FUNCTION_BLOCK FB_V1_C1_Virtual_Input_Source IMPLEMENTS I_VirtualInputSource, I_V1_Virtual_Input_Source
VAR
	_fbSource: I_InputSource;
	
	_nSourceClientID: LWORD;
	_nDataHandle: ULINT;
	_nElements: UDINT;
	
	_nSelectedElement: UDINT;
	_nSelectedOversample: UDINT;
	
	_nContext: DWORD;
	_stInputs: ST_T1_Inputs;
	
	_nTimestamp: ULINT;
END_VAR

PROPERTY bEndOfData : BOOL
GET
bEndOfData:= _nElements = 0 OR (_nSelectedElement >= _nElements AND _nSelectedOversample >= _fbSource.nMaxOversamplingFactor);
END_GET
END_PROPERTY

METHOD Done : BOOL
VAR
END_VAR
IF bEndOfData AND _nElements > 0 THEN
	_nElements:= 0;
	_fbSource.ClientDone(_nSourceClientID);
END_IF

_nContext:= 0;
END_METHOD

PROPERTY dtTimestamp : DCTIMESTRUCT
GET
dtTimestamp:= F_AlyTimestampToDCTimestruct(_nTimestamp);
END_GET
END_PROPERTY

PROPERTY eSourceState : E_DataSourceState
GET
eSourceState:= _fbSource.eDataState;
END_GET
END_PROPERTY

METHOD FB_init : BOOL
VAR_INPUT
	bInitRetains: BOOL; // if TRUE, the retain variables are initialized (warm start / cold start)
	bInCopyCode: BOOL; // if TRUE, the instance afterwards gets moved into the copy code (online change)
	fbSource: I_InputSource;
END_VAR
VAR
END_VAR
IF NOT bInCopyCode THEN
	fbSource.AddClient(nClientID=>_nSourceClientID);
	_fbSource:= fbSource;
END_IF
END_METHOD

PROPERTY fbInputSource : I_InputSource
GET
fbInputSource:= _fbSource;
END_GET
END_PROPERTY

PROPERTY nContext : DWORD
GET
nContext:= _nContext;
END_GET
END_PROPERTY

PROPERTY nDataHandle : ULINT
GET
nDataHandle:= _nDataHandle;
END_GET
END_PROPERTY

METHOD NextData : BOOL
VAR_INPUT
	nMaxOversampling: UDINT;
END_VAR
VAR
END_VAR
IF _nElements > 0 AND NOT bEndOfData THEN

	_nSelectedOversample:= _nSelectedOversample + 1;
	IF _nSelectedOversample > nMaxOversampling OR _nSelectedElement = 0 THEN
		_nSelectedElement:= _nSelectedElement + 1;
		_nSelectedOversample:= 1;
	END_IF

	NextData:= _fbSource.GetData(_nSelectedElement, ADR(_stInputs), SIZEOF(_stInputs), nTimestamp=>_nTimestamp, nContext=>_nContext);
	_nContext:= _nContext OR E_VirtualInput.eContext_V1_Virtual_Input_Source;
END_IF
END_METHOD

PROPERTY nV1_nDefectiveUnits : ULINT
GET
nV1_nDefectiveUnits:= _stInputs.nGVL_Components_fbMachine_stAnalytics_nDefectiveUnits;
END_GET
END_PROPERTY

PROPERTY nV1_nState : UINT
GET
nV1_nState:= _stInputs.nGVL_Components_fbMachine_stAnalytics_nState;
END_GET
END_PROPERTY

PROPERTY nV1_nUnitsProduced : ULINT
GET
nV1_nUnitsProduced:= _stInputs.nGVL_Components_fbMachine_stAnalytics_nUnitsProduced;
END_GET
END_PROPERTY

PROPERTY nV1_tMlCalculation : UDINT
GET
nV1_tMlCalculation:= _stInputs.nGVL_Components_fbMachine_stAnalytics_tMlCalculation;
END_GET
END_PROPERTY

METHOD SourceSync : BOOL
VAR
END_VAR
IF _fbSource.NewDataAvailable(_nDataHandle) THEN
	_nDataHandle:= _fbSource.nDataHandle;
	_nElements:= _fbSource.nElements;

	_nSelectedElement:= 0;
	_nSelectedOversample:= 0;
END_IF
END_METHOD

PROPERTY tTimestamp : ULINT
GET
tTimestamp:= _nTimestamp;
END_GET
END_PROPERTY

END_FUNCTION_BLOCK

(* stored: Version 1.2.0.0, ProductVersion 3.1.4024.13
   POU FB_V1_C1_Virtual_Input_Source: Id {9a6257cd-c1e8-4e82-8d92-73bc8f8dbf80}, SpecialFunc None
   Folder I_V1_Virtual_Input_Source: Id {efc72da7-a840-4c18-9a1b-93ce3ac4e1a4}
   Folder I_VirtualInputSource: Id {bb4f3988-481a-4578-816a-057dfc1780de}
   Property bEndOfData: Id {5a4d4dd8-e514-462b-bbe9-2121c90468f9}
   Get Get: Id {7d2674b7-e798-47c8-8c4a-7094fac53df9}
   Method Done: Id {77b24883-a059-45f4-8b35-6973e05288f8}
   Property dtTimestamp: Id {400a5cc9-42de-4db8-9375-3e39e2975a34}
   Get Get: Id {d595a4e9-9059-4ab6-bcab-c824b16b2ab1}
   Property eSourceState: Id {3fadf5ac-338e-4bac-a55c-43fada65f2a8}
   Get Get: Id {9906be45-3dc9-4007-890c-00020d9d677c}
   Method FB_init: Id {84d9821c-cc28-48b6-8dab-7a1f061061a9}
   Property fbInputSource: Id {b3611652-af3f-4039-807a-6015d990d91b}
   Get Get: Id {96e89225-b1a3-47ba-8433-72c177d3226c}
   Property nContext: Id {588a0dcc-cb20-4e63-9a97-282e0f27c55b}
   Get Get: Id {090de91a-e787-4045-aa95-0a3d47490d4f}
   Property nDataHandle: Id {38c2699e-da6d-4c1b-8d7b-2604eadc34ec}
   Get Get: Id {85a89889-8df5-433e-9a6b-a2f7693df06d}
   Method NextData: Id {e2348384-aa9f-4400-9db6-bcb1ae420b6e}
   Property nV1_nDefectiveUnits: Id {6e202291-3174-4e5b-a9b1-0ff2b2499ade}
   Get Get: Id {f25bd935-c88e-4c8a-b9e7-b464fcf61026}
   Property nV1_nState: Id {87e07056-3e7e-493d-bd12-ce306d4fa93a}
   Get Get: Id {d72da6c5-df2b-4e49-87b7-3179248a3f84}
   Property nV1_nUnitsProduced: Id {fc9e88c7-34c1-49ca-be27-2ed51d12776d}
   Get Get: Id {4c8e876b-9bdf-4651-89cc-2b92fa67cd62}
   Property nV1_tMlCalculation: Id {0cfeb22c-47b7-410d-8580-7225c8318356}
   Get Get: Id {582aef3e-93de-4b0a-a8a2-6d5424920887}
   Method SourceSync: Id {facef239-7c06-4502-93b6-2ae10d200b44}
   Property tTimestamp: Id {e6a49db7-eb8c-499a-9c3f-98e9179ed2b6}
   Get Get: Id {8a0269aa-384e-498a-a1ca-4dbf295766f9} *)
